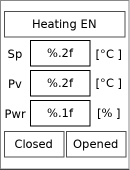
VISUALIZATION vHP3_HeatedPlateData  // 130x170
VAR_IN_OUT
	fbHP	: fbHPv3_Control;
END_VAR
    RoundedRectangle (0,0 129x170)
    Rectangle (30,40 60x26), "%.2f", text variable: fbHP.fbHP_PID.SET_POINT
    Label (94,41 30x26), "[°C ]"
    Label (0,41 30x26), "Sp"
    Rectangle (30,70 60x26), "%.2f", text variable: fbHP.fbHP_PID.ACTUAL
    Label (94,70 30x26), "[°C ]"
    Label (0,71 30x26), "Pv"
    Rectangle (30,100 60x26), "%.1f", text variable: fbHP.rHPHeaterPower
    Label (94,100 30x26), "[% ]"
    Label (0,101 30x26), "Pwr"
    Rectangle (4,131 60x26), "Closed", colour toggle: fbHP.fbHeatedPlate_Actuator.Closed
    Rectangle (66,131 60x26), "Opened", colour toggle: fbHP.fbHeatedPlate_Actuator.Opened
    Rectangle (4,11 121x26), "Heating EN", colour toggle: fbHP.fbHP_HeaterON.Q
END_VISUALIZATION

(* stored: Version 1.1.0.1, ProductVersion 3.1.4024.12
   Visu vHP3_HeatedPlateData: Id {31b396fc-aca8-46d1-b0df-cacaceca3a98} *)
